KUKA KRL program: masref_user.src, masref_user.dat

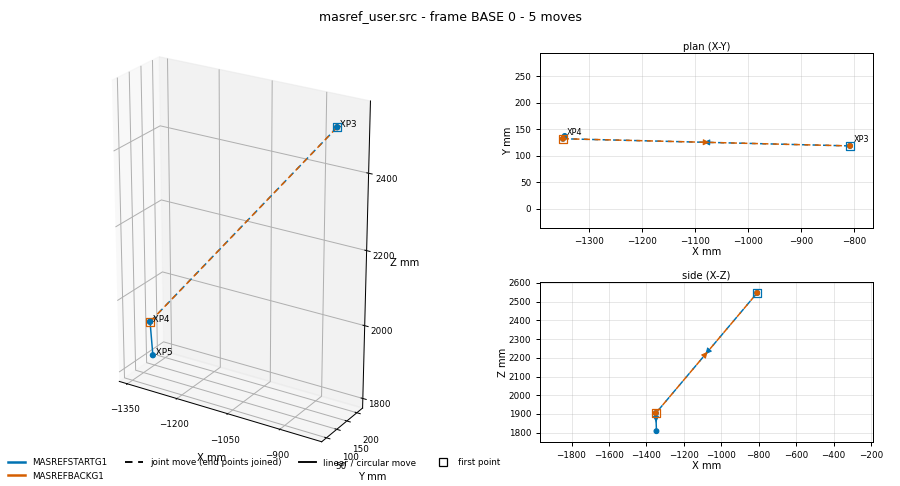
[picture p0: tool path of masref_user.src in frame BASE 0, 5 of 6 moves have a stored position in this frame; points joined in program order, loops and branches not executed]
--- masref_user.src ---
&ACCESS RVO26
&REL 12
&COMMENT Mastering Reference User Program
&PARAM DISKPATH = KRC:\R1\Program
DEF MasRef_USER()
END

GLOBAL DEF MASREFSTARTG1()
;FOLD Teach path and position for reference group 1
;ENDFOLD


;FOLD PTP P3 CONT Vel=100 % PDAT3 Tool[8]:TOOL_CHANGER Base[0];%{PE}%R 8.2.20,%MKUKATPBASIS,%CMOVE,%VPTP,%P 1:PTP, 2:P3, 3:C_DIS, 5:100, 7:PDAT3
$BWDSTART=FALSE
PDAT_ACT=PPDAT3
FDAT_ACT=FP3
BAS(#PTP_PARAMS,100)
PTP XP3 C_DIS
;ENDFOLD
;FOLD PTP P4 CONT Vel=100 % PDAT4 Tool[8]:TOOL_CHANGER Base[0];%{PE}%R 8.2.20,%MKUKATPBASIS,%CMOVE,%VPTP,%P 1:PTP, 2:P4, 3:C_DIS, 5:100, 7:PDAT4
$BWDSTART=FALSE
PDAT_ACT=PPDAT4
FDAT_ACT=FP4
BAS(#PTP_PARAMS,100)
PTP XP4 C_DIS
;ENDFOLD

;FOLD LIN P5 Vel=0.5 m/s CPDAT3 Tool[8]:TOOL_CHANGER Base[0];%{PE}%R 8.2.20,%MKUKATPBASIS,%CMOVE,%VLIN,%P 1:LIN, 2:P5, 3:, 5:0.5, 7:CPDAT3
$BWDSTART=FALSE
LDAT_ACT=LCPDAT3
FDAT_ACT=FP5
BAS(#CP_PARAMS,0.5)
LIN XP5
;ENDFOLD

END

GLOBAL DEF MASREFBACKG1()
;FOLD Teach path back for reference group 1
;ENDFOLD


;FOLD PTP P6 CONT Vel=100 % PDAT5 Tool[8]:TOOL_CHANGER Base[0];%{PE}%R 8.2.20,%MKUKATPBASIS,%CMOVE,%VPTP,%P 1:PTP, 2:P6, 3:C_DIS, 5:100, 7:PDAT5
$BWDSTART=FALSE
PDAT_ACT=PPDAT5
FDAT_ACT=FP6
BAS(#PTP_PARAMS,100)
PTP XP6 C_DIS
;ENDFOLD
;FOLD PTP P7 CONT Vel=100 % PDAT6 Tool[8]:TOOL_CHANGER Base[0];%{PE}%R 8.2.20,%MKUKATPBASIS,%CMOVE,%VPTP,%P 1:PTP, 2:P7, 3:C_DIS, 5:100, 7:PDAT6
$BWDSTART=FALSE
PDAT_ACT=PPDAT6
FDAT_ACT=FP7
BAS(#PTP_PARAMS,100)
PTP XP7 C_DIS
;ENDFOLD

;FOLD PTP HOME Vel=100 % DEFAULT;%{PE}%R 8.2.20,%MKUKATPBASIS,%CMOVE,%VPTP,%P 1:PTP, 2:HOME, 3:, 5:100, 7:DEFAULT
$BWDSTART=FALSE
PDAT_ACT=PDEFAULT
FDAT_ACT=FHOME
BAS(#PTP_PARAMS,100)
$H_POS=XHOME
PTP XHOME
;ENDFOLD


END

GLOBAL DEF MASREFSTARTG2()
;FOLD Teach path and position for reference group 2
;ENDFOLD

END

GLOBAL DEF MASREFBACKG2()
;FOLD Teach path back for reference group 2
;ENDFOLD

END

GLOBAL DEF MASREFSTARTG3()
;FOLD Teach path and position for reference group 3
;ENDFOLD

END

GLOBAL DEF MASREFBACKG3()
;FOLD Teach path back for reference group 3
;ENDFOLD

END

--- masref_user.dat ---
&ACCESS RVO26
&REL 12
&COMMENT Mastering Reference User Program
&PARAM DISKPATH = KRC:\R1\Program
DEFDAT  masref_user
;FOLD EXTERNAL DECLARATIONS;%{PE}%MKUKATPBASIS,%CEXT,%VCOMMON,%P
;FOLD GRIPPERTECH EXT
EXT  H50 (INT  :IN,INT  :IN,INT  :IN,GRP_TYP  :IN )
;ENDFOLD (GRIPPERTECH EXT)
;FOLD SPOTTECH EXT
EXT  USERSPOT (S_COMMAND  :IN,SPOT_TYPE  :IN )
;ENDFOLD (SPOTTECH EXT)
;FOLD BASISTECH EXT;%{PE}%MKUKATPBASIS,%CEXT,%VEXT,%P
EXT  BAS (BAS_COMMAND  :IN,REAL  :IN )
;ENDFOLD (BASISTECH EXT)
;FOLD USER EXT;%{E}%MKUKATPUSER,%CEXT,%VEXT,%P
;Make here your modifications

;ENDFOLD (USER EXT)
;ENDFOLD (EXTERNAL DECLERATIONS)
DECL BASIS_SUGG_T LAST_BASIS={POINT1[] "P0                      ",POINT2[] "P0                      ",CP_PARAMS[] "CPDAT0                  ",PTP_PARAMS[] "PDAT0                   ",CONT[] "                        ",CP_VEL[] "2.0                     ",PTP_VEL[] " 100                    ",SYNC_PARAMS[] "SYNCDAT                 ",SPL_NAME[] "S0                      "}
DECL PDAT PPDAT3={VEL 100.0,ACC 100.0,APO_DIST 100.0,APO_MODE #CDIS}
DECL E6POS XP3={X -808.14801,Y 118.585999,Z 2546.57104,A 58.656189,B -15.01828,C -153.726593,S 2,T 3,E1 -1221.89294,E2 0.0,E3 0.0,E4 0.0,E5 0.0,E6 0.0}
DECL FDAT FP3={TOOL_NO 8,BASE_NO 0,IPO_FRAME #BASE,POINT2[] " ",TQ_STATE FALSE}
DECL PDAT PPDAT4={VEL 100.0,ACC 100.0,APO_DIST 25.0,APO_MODE #CDIS}
DECL E6POS XP4={X -1349.40002,Y 132.080505,Z 1904.422,A 103.248596,B -7.45883703,C -175.902695,S 2,T 11,E1 -1536.41394,E2 0.0,E3 0.0,E4 0.0,E5 0.0,E6 0.0}
DECL FDAT FP4={TOOL_NO 8,BASE_NO 0,IPO_FRAME #BASE,POINT2[] " ",TQ_STATE FALSE}
DECL LDAT LCPDAT3={VEL 2.0,ACC 100.0,APO_DIST 100.0,APO_FAC 50.0,AXIS_VEL 100.0,AXIS_ACC 100.0,ORI_TYP #VAR,CIRC_TYP #BASE,JERK_FAC 50.0,GEAR_JERK 50.0,EXAX_IGN 0}
DECL E6POS XP5={X -1346.15198,Y 137.332108,Z 1807.93896,A 107.038101,B -14.0545502,C 175.665802,S 2,T 3,E1 -1522.88306,E2 0.0,E3 0.0,E4 0.0,E5 0.0,E6 0.0}
DECL FDAT FP5={TOOL_NO 8,BASE_NO 0,IPO_FRAME #BASE,POINT2[] " ",TQ_STATE FALSE}
DECL PDAT PPDAT5={VEL 100.0,ACC 100.0,APO_DIST 100.0,APO_MODE #CDIS}
DECL E6POS XP6={X -1349.41602,Y 132.136993,Z 1904.44397,A 103.212898,B -7.7540369,C -171.195801,S 2,T 11,E1 -1536.40405,E2 0.0,E3 0.0,E4 0.0,E5 0.0,E6 0.0}
DECL FDAT FP6={TOOL_NO 8,BASE_NO 0,IPO_FRAME #BASE,POINT2[] " ",TQ_STATE FALSE}
DECL PDAT PPDAT6={VEL 100.0,ACC 100.0,APO_DIST 100.0,APO_MODE #CDIS}
DECL E6POS XP7={X -808.14801,Y 118.585999,Z 2546.57104,A 58.656189,B -15.01828,C -153.726593,S 2,T 3,E1 -1221.89294,E2 0.0,E3 0.0,E4 0.0,E5 0.0,E6 0.0}
DECL FDAT FP7={TOOL_NO 8,BASE_NO 0,IPO_FRAME #BASE,POINT2[] " ",TQ_STATE FALSE}
ENDDAT
